// TIA Portal project "Comparadores" (V16)

(* hardware
DEVICE "S7-1200 station_1"  S7-1200 Station
   slot 0: "Rack_0"  S7-1200 Rack  Rack  V1.0
   slot 1: "PLC_1"  CPU 1214C AC/DC/Rly  6ES7 214-1BG40-0XB0  V4.4
*)

// ===== PLC "PLC_1"  CPU 1214C AC/DC/Rly =====

VAR_GLOBAL   // PLC tag table "Tabla de variables estándar"
   "INT TMP" AT %I0.0 : Bool;
   "MEMORIA TEMPO" AT %MD105 : Time;
   "INT CU" AT %I0.1 : Bool;
   "INT CD" AT %I0.2 : Bool;
   "INT RESET UP" AT %I0.3 : Bool;
   "INT RESET DOWN" AT %I0.4 : Bool;
   "MEMORIA CTUD" AT %MW101 : Int;
   "CONTACTO NC" AT %I0.5 : Bool;
   "Tag_2" AT %Q0.0 : Bool;
   "Tag_3" AT %Q0.1 : Bool;
   "Tag_1" AT %Q0.2 : Bool;
   "Tag_4" AT %Q0.3 : Bool;
   "Tag_5" AT %Q0.4 : Bool;
   "Tag_6" AT %Q0.5 : Bool;
   "Tag_7" AT %Q0.6 : Bool;
   "Tag_8" AT %MW10 : Int;
   "Tag_9" AT %MD200 : Real;
   "Tag_10" AT %Q0.7 : Bool;
   "Tag_11" AT %Q1.0 : Bool;
   "Tag_12" AT %MD201 : Real;
END_VAR

// folder: System blocks/Program resources

DATA_BLOCK "IEC_Timer_0_DB"   // DB1
{ S7_Optimized_Access := 'TRUE' }
AUTHOR : Simatic
FAMILY : IEC
NAME : IEC_TMR
VERSION : 1.0
// stored: InstanceOfName IEC_TIMER
"IEC_TIMER"
BEGIN
END_DATA_BLOCK

DATA_BLOCK "IEC_Counter_0_DB"   // DB2
{ S7_Optimized_Access := 'TRUE' }
AUTHOR : Simatic
FAMILY : IEC
NAME : CNTR
VERSION : 1.0
// stored: InstanceOfName IEC_COUNTER
"IEC_COUNTER"
BEGIN
END_DATA_BLOCK

// folder: (top level)

ORGANIZATION_BLOCK "Main"   // OB1, LAD, ProgramCycle
TITLE = "Main Program Sweep (Cycle)"
{ S7_Optimized_Access := 'TRUE' }
VERSION : 0.1
   VAR_INPUT
      Initial_Call : Bool;   // Initial call of this OB
      Remanence : Bool;   // =True, if remanent data are available
   END_VAR
BEGIN

REGION Network 1
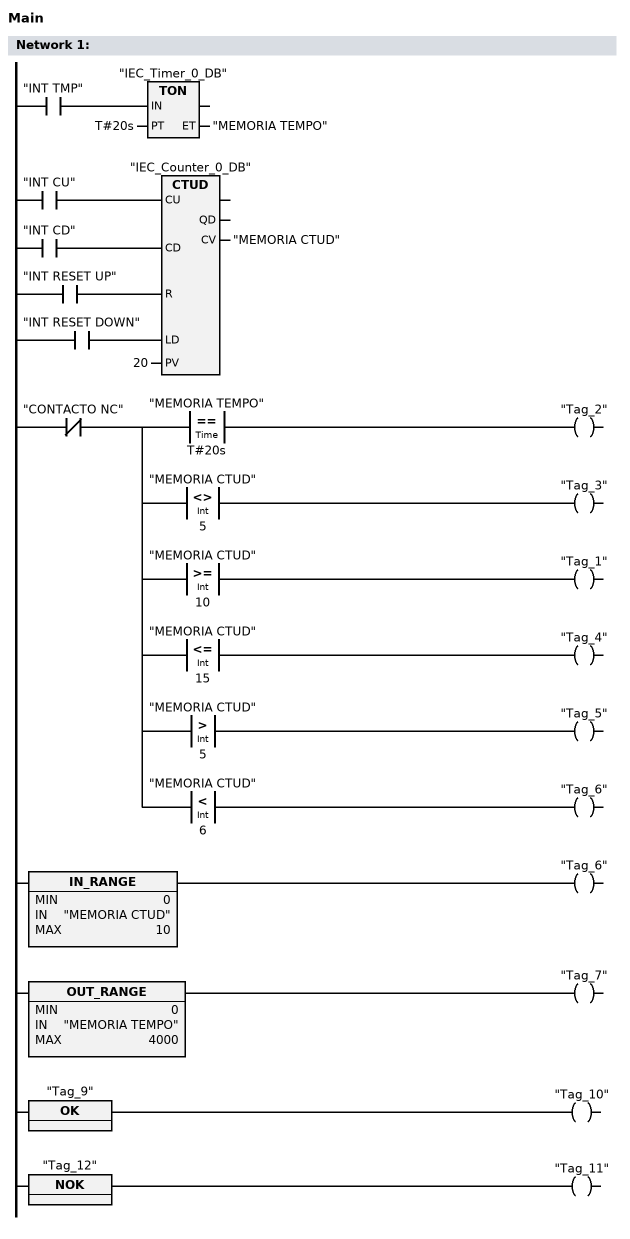
   // no SCL statement known for NOK, OK: written as a call
   "IEC_Timer_0_DB".TON(IN := "INT TMP", PT := T#20s, ET => "MEMORIA TEMPO");
   "IEC_Counter_0_DB".CTUD(CU := "INT CU",
                           CD := "INT CD",
                           R := "INT RESET UP",
                           LD := "INT RESET DOWN",
                           PV := 20,
                           CV => "MEMORIA CTUD");
   "Tag_2" := NOT "CONTACTO NC" AND ("MEMORIA TEMPO" = T#20s);
   "Tag_3" := NOT "CONTACTO NC" AND ("MEMORIA CTUD" <> 5);
   "Tag_1" := NOT "CONTACTO NC" AND ("MEMORIA CTUD" >= 10);
   "Tag_4" := NOT "CONTACTO NC" AND ("MEMORIA CTUD" <= 15);
   "Tag_5" := NOT "CONTACTO NC" AND ("MEMORIA CTUD" > 5);
   "Tag_6" := NOT "CONTACTO NC" AND ("MEMORIA CTUD" < 6);
   "Tag_6" := (0 <= "MEMORIA CTUD") AND ("MEMORIA CTUD" <= 10);
   "Tag_7" := ("MEMORIA TEMPO" < 0) OR ("MEMORIA TEMPO" > 4000);
   "Tag_10" := OK("Tag_9");
   "Tag_11" := NOK("Tag_12");
END_REGION
END_ORGANIZATION_BLOCK